// TIA Portal V19 export
TYPE "IPC_Msg_Log_PAR"
   STRUCT
      Id : DInt;   // Identificativo progressivo univoco del messaggio (0 = cella vuota)
      timestamp : String;   // Timestamp evento formato ISO: YYYY-MM-DD HH:MM:SS.mmm
      topic : UDInt;   // Categoria/argomento del log per filtering e routing.
      payLoad_1 : String;   // Record di valori [ScreenNumber/RowNumber]=Value;
      payLoad_2 : String;   // Record di valori [ScreenNumber/RowNumber]=Value;
      payLoad_3 : String;   // Record di valori [ScreenNumber/RowNumber]=Value;
      payLoad_4 : String;   // Record di valori [ScreenNumber/RowNumber]=Value;
      payLoad_5 : String;   // Record di valori [ScreenNumber/RowNumber]=Value;
   END_STRUCT;
END_TYPE
